TYPE ST_HMI_Monitor_FireDetection :
STRUCT
	e_SmokeDetectorState			: eSmokeDetectAlarmStatus;
	e_CoDetectorState				: eCOAlarmStatus;
	r_CoDetectorLeftValue			: REAL; //ppm
	r_CoDetectorRightValue			: REAL; //ppm			
END_STRUCT
END_TYPE

(* stored: Version 1.1.0.1, ProductVersion 3.1.4026.18
   DUT ST_HMI_Monitor_FireDetection: Id {b1c8f49e-f4b4-4d94-a6a3-facc1588d496} *)
